(* IEC 61131-3 sources: A_BST22/ (part 2) *)

(* ---- simon_says_ladder_logic.st ---- *)
(*
Simon Says Game - Ladder Logic Implementation
Phase 1: 3 Buttons (Red, Blue, Yellow)
For Omron NX102-1100 PLC with Sysmac Studio

Author: Assistant
Date: 2025-10-01
Version: 1.0
*)

PROGRAM SimonSaysGame
VAR
    // Local working variables
    i : INT;
    ButtonPressed : INT;
    SequenceMatch : BOOL;
END_VAR

(* ========================================
   RUNG 1: INPUT MAPPING AND EDGE DETECTION
   ======================================== *)

// Map physical inputs to variables
RedButton_Input := %IX0.5;      // DI5
BlueButton_Input := %IX0.3;     // DI3
YellowButton_Input := %IX0.1;   // DI1

// Edge detection for button presses
RedButton_Rising := RedButton_Input AND NOT RedButton_Prev;
BlueButton_Rising := BlueButton_Input AND NOT BlueButton_Prev;
YellowButton_Rising := YellowButton_Input AND NOT YellowButton_Prev;

// Store previous states
RedButton_Prev := RedButton_Input;
BlueButton_Prev := BlueButton_Input;
YellowButton_Prev := YellowButton_Input;

(* ========================================
   RUNG 2: GAME INITIALIZATION
   ======================================== *)

// Initialize game on first scan or reset
IF FIRST_SCAN OR GameReset THEN
    GameState := 0;             // Idle state
    GameActive := FALSE;
    CurrentLevel := 1;
    SequenceLength := 1;
    PlaybackIndex := 0;
    InputIndex := 1;
    GameReset := FALSE;

    // Clear sequence array
    FOR i := 1 TO MaxLevel DO
        GameSequence[i] := 0;
    END_FOR;

    // Initialize random seed with system time
    RandomSeed := DWORD_TO_TIME(TIME());
END_IF;

(* ========================================
   RUNG 3: GAME START TRIGGER
   ======================================== *)

// Start game when any button is pressed in idle state
IF GameState = 0 AND (RedButton_Rising OR BlueButton_Rising OR YellowButton_Rising) THEN
    GameState := 1;             // Generate new sequence
    GameActive := TRUE;
    CurrentLevel := 1;
    SequenceLength := 1;
    GameWon := FALSE;
    GameLost := FALSE;
END_IF;

(* ========================================
   RUNG 4: RANDOM SEQUENCE GENERATION
   ======================================== *)

// Generate new sequence element
IF GameState = 1 THEN
    // Simple linear congruential generator for random numbers
    RandomValue := (RandomSeed * 1103515245 + 12345) MOD 16#7FFFFFFF;
    RandomSeed := RandomValue;

    // Convert to button number (1=Red, 2=Blue, 3=Yellow)
    NextButton := (INT(RandomValue MOD 3)) + 1;

    // Add to sequence
    GameSequence[SequenceLength] := NextButton;

    // Move to playback state
    GameState := 2;
    PlaybackIndex := 1;
    PlaybackActive := TRUE;

    // Start first flash timer
    FlashTimer.IN := TRUE;
    FlashTimer.PT := FLASH_TIME;
END_IF;

(* ========================================
   RUNG 5: SEQUENCE PLAYBACK LOGIC
   ======================================== *)

// Handle LED flashing during playback
IF GameState = 2 AND PlaybackActive THEN

    // Flash current button in sequence
    CASE GameSequence[PlaybackIndex] OF
        1: RedLED_Output := FlashTimer.IN AND NOT FlashTimer.Q;      // Red
        2: BlueLED_Output := FlashTimer.IN AND NOT FlashTimer.Q;     // Blue
        3: YellowLED_Output := FlashTimer.IN AND NOT FlashTimer.Q;   // Yellow
    END_CASE;

    // When flash timer expires, start gap timer
    IF FlashTimer.Q THEN
        FlashTimer.IN := FALSE;
        GapTimer.IN := TRUE;
        GapTimer.PT := GAP_TIME;

        // Turn off all LEDs during gap
        RedLED_Output := FALSE;
        BlueLED_Output := FALSE;
        YellowLED_Output := FALSE;
    END_IF;

    // When gap timer expires, move to next button or finish playback
    IF GapTimer.Q THEN
        GapTimer.IN := FALSE;
        PlaybackIndex := PlaybackIndex + 1;

        IF PlaybackIndex > SequenceLength THEN
            // Playback complete, start input phase
            PlaybackActive := FALSE;
            GameState := 3;
            InputIndex := 1;
            InputTimer.IN := TRUE;
            InputTimer.PT := INPUT_TIMEOUT;
        ELSE
            // Start next flash
            FlashTimer.IN := TRUE;
            FlashTimer.PT := FLASH_TIME;
        END_IF;
    END_IF;
END_IF;

// Call timer function blocks
FlashTimer();
GapTimer();

(* ========================================
   RUNG 6: PLAYER INPUT HANDLING
   ======================================== *)

// Handle player input during input phase
IF GameState = 3 THEN

    // Determine which button was pressed
    ButtonPressed := 0;
    IF RedButton_Rising THEN
        ButtonPressed := 1;
        LastButtonPressed := 1;
    ELSIF BlueButton_Rising THEN
        ButtonPressed := 2;
        LastButtonPressed := 2;
    ELSIF YellowButton_Rising THEN
        ButtonPressed := 3;
        LastButtonPressed := 3;
    END_IF;

    // Process button press
    IF ButtonPressed > 0 THEN
        // Check if correct button
        IF ButtonPressed = GameSequence[InputIndex] THEN
            CorrectSequence := TRUE;
            InputIndex := InputIndex + 1;

            // Reset input timer for next button
            InputTimer.IN := FALSE;
            InputTimer.IN := TRUE;
            InputTimer.PT := INPUT_TIMEOUT;

            // Check if sequence complete
            IF InputIndex > SequenceLength THEN
                // Level complete!
                GameState := 4;  // Success state
                SuccessTimer.IN := TRUE;
                SuccessTimer.PT := SUCCESS_DELAY;
            END_IF;
        ELSE
            // Wrong button - game over
            CorrectSequence := FALSE;
            GameState := 5;  // Fail state
            GameLost := TRUE;
        END_IF;
    END_IF;

    // Check for input timeout
    IF InputTimer.Q THEN
        GameState := 5;  // Fail state
        GameLost := TRUE;
        InputTimeout := TRUE;
    END_IF;

    InputTimer();
END_IF;

(* ========================================
   RUNG 7: SUCCESS HANDLING
   ======================================== *)

// Handle successful level completion
IF GameState = 4 THEN

    // Flash all LEDs to indicate success
    RedLED_Output := TRUE;
    BlueLED_Output := TRUE;
    YellowLED_Output := TRUE;

    // When success timer expires, advance to next level
    IF SuccessTimer.Q THEN
        SuccessTimer.IN := FALSE;
        CurrentLevel := CurrentLevel + 1;
        SequenceLength := SequenceLength + 1;

        // Check if game won (max level reached)
        IF CurrentLevel > MaxLevel THEN
            GameWon := TRUE;
            GameState := 0;  // Return to idle
            GameActive := FALSE;
        ELSE
            // Generate next level
            GameState := 1;
        END_IF;

        // Turn off success LEDs
        RedLED_Output := FALSE;
        BlueLED_Output := FALSE;
        YellowLED_Output := FALSE;
    END_IF;

    SuccessTimer();
END_IF;

(* ========================================
   RUNG 8: FAILURE HANDLING
   ======================================== *)

// Handle game failure
IF GameState = 5 THEN

    // Flash all LEDs rapidly to indicate failure
    IF (TIME() MOD T#200ms) < T#100ms THEN
        RedLED_Output := TRUE;
        BlueLED_Output := TRUE;
        YellowLED_Output := TRUE;
    ELSE
        RedLED_Output := FALSE;
        BlueLED_Output := FALSE;
        YellowLED_Output := FALSE;
    END_IF;

    // Auto-reset after 3 seconds
    IF NOT SuccessTimer.IN THEN
        SuccessTimer.IN := TRUE;
        SuccessTimer.PT := T#3000ms;
    END_IF;

    IF SuccessTimer.Q THEN
        GameReset := TRUE;
        SuccessTimer.IN := FALSE;
    END_IF;

    SuccessTimer();
END_IF;

(* ========================================
   RUNG 9: OUTPUT MAPPING
   ======================================== *)

// Map LED outputs to physical outputs
%QX0.0 := RedLED_Output;        // DO0
%QX0.1 := BlueLED_Output;       // DO1
%QX0.2 := YellowLED_Output;     // DO2

(* ========================================
   RUNG 10: STATUS AND DEBUG
   ======================================== *)

// Update debug status string
CASE GameState OF
    0: DebugState := 'IDLE - Press any button to start';
    1: DebugState := 'GENERATING sequence';
    2: DebugState := 'PLAYBACK - Watch the sequence';
    3: DebugState := 'INPUT - Repeat the sequence';
    4: DebugState := 'SUCCESS - Level complete!';
    5: DebugState := 'FAILED - Game over';
END_CASE;

// Test mode - all LEDs on (for testing)
IF AllLEDs_Test THEN
    %QX0.0 := TRUE;  // Red LED
    %QX0.1 := TRUE;  // Blue LED
    %QX0.2 := TRUE;  // Yellow LED
END_IF;

END_PROGRAM

(* ---- SimonSays.st ---- *)
// MAIN is N.C. → LED on when pressed
OLED_MAIN := NOT IBTN_MAIN;

// Color buttons → LED (when not in sequence display mode)
IF NOT SeqDisplay_Active THEN
    OLED_B := IBTN_B;
    OLED_R := IBTN_R;
    OLED_Y := IBTN_Y;
END_IF;

//  main game logic
Trig_Start(Clk := IBTN_B, Q => B);

IF B THEN
    Rand_Gen(Execute := TRUE, Seed := 0, Rnd => RandN);

    IF RandN < 0.333 THEN
        L_N := 1;  // Yellow
    ELSIF RandN < 0.666 THEN
        L_N := 2;  // Blue
    ELSE
        L_N := 3;  // Red
    END_IF;

    IF WriteIndex >= 50 THEN
        WriteIndex := 0;
        ArrayFull := TRUE;
    ELSIF WriteIndex < 0 THEN
        WriteIndex := 0;
    END_IF;

    Idx := TO_INT(WriteIndex);
    GameFlow_SN[Idx] := L_N;
    WriteIndex := WriteIndex + 1;

    // Trigger sequence display after adding new number
    SeqDisplay_Active := TRUE;
    SeqDisplay_Index := 0;
    SeqDisplay_Step := 0;  // 0 = LED ON, 1 = LED OFF
    T_SeqDisplay(IN := FALSE, PT := T#300ms);
END_IF;

// --- Sequence Display Logic ---
IF SeqDisplay_Active THEN
    IF NOT T_SeqDisplay.Q THEN
        T_SeqDisplay(IN := TRUE, PT := T#300ms);
    ELSE
        T_SeqDisplay(IN := FALSE, PT := T#300ms);
    END_IF;

    Trig_SeqTick(CLK := T_SeqDisplay.Q);
    SeqDisplay_Tick := Trig_SeqTick.Q;

    IF SeqDisplay_Tick THEN
        IF SeqDisplay_Step = 0 THEN
            // LED ON - display current sequence element
            CASE GameFlow_SN[SeqDisplay_Index] OF
                1:  OLED_Y := TRUE;  OLED_B := FALSE; OLED_R := FALSE;  // Yellow
                2:  OLED_Y := FALSE; OLED_B := TRUE;  OLED_R := FALSE;  // Blue
                3:  OLED_Y := FALSE; OLED_B := FALSE; OLED_R := TRUE;   // Red
                ELSE
                    OLED_Y := FALSE; OLED_B := FALSE; OLED_R := FALSE;
            END_CASE;
            SeqDisplay_Step := 1;
        ELSE
            // LED OFF - pause between elements
            OLED_Y := FALSE; OLED_B := FALSE; OLED_R := FALSE;
            SeqDisplay_Step := 0;
            SeqDisplay_Index := SeqDisplay_Index + 1;

            // Check if we've displayed the entire sequence
            IF SeqDisplay_Index >= WriteIndex THEN
                SeqDisplay_Active := FALSE;
                OLED_Y := FALSE; OLED_B := FALSE; OLED_R := FALSE;
            END_IF;
        END_IF;
    END_IF;
END_IF;

// -auto-reset edge when WriteIndex hits 50
Trig_Wrap(CLK := (WriteIndex = 50));
ResetReq := RI OR Trig_Wrap.Q;      // manual RI or auto edge at 50
Trig_Reset(CLK := ResetReq);

IF Trig_Reset.Q THEN
    AryAddV(In1 := GameFlow_S[0], In2 := L_N, Size := 50, AryOut := GameFlow_SN[0]);

    GameOver_Active := TRUE;
    GameOver_Step := -1;
    T_Seq(IN := FALSE, PT := T#300ms);

    WriteIndex := 0;
    ArrayFull := TRUE;
END_IF;

// --- game over LED sequence (R -> B -> Y, once) ---
IF GameOver_Active THEN
    IF NOT T_Seq.Q THEN
        T_Seq(IN := TRUE, PT := T#300ms);
    ELSE
        T_Seq(IN := FALSE, PT := T#300ms);
    END_IF;

    Trig_Tick(CLK := T_Seq.Q);
    GameOver_Tick := Trig_Tick.Q;

    IF GameOver_Tick THEN
        GameOver_Step := GameOver_Step + 1;
    END_IF;

    CASE GameOver_Step OF
        0:  OLED_R := TRUE;  OLED_B := FALSE; OLED_Y := FALSE;
        1:  OLED_R := FALSE; OLED_B := TRUE;  OLED_Y := FALSE;
        2:  OLED_R := FALSE; OLED_B := FALSE; OLED_Y := TRUE;
        4:  OLED_R := FALSE; OLED_B := FALSE; OLED_Y := FALSE;
        5:  OLED_R := TRUE;  OLED_B := TRUE;  OLED_Y := TRUE;
        6:  OLED_R := FALSE; OLED_B := FALSE; OLED_Y := FALSE;
        7:  OLED_R := TRUE;  OLED_B := TRUE;  OLED_Y := TRUE;
        ELSE
            OLED_R := FALSE; OLED_B := FALSE; OLED_Y := FALSE;
    END_CASE;

    IF GameOver_Step > 7 THEN
        GameOver_Active := FALSE;
        OLED_R := FALSE; OLED_B := FALSE; OLED_Y := FALSE;
    END_IF;
END_IF;

(* ---- SimonSays_Phase1.st ---- *)
(* ====================================================================
   SIMON SAYS GAME - PHASE 1 (3 BUTTONS)
   For Omron NX102-1100 PLC

   Hardware Configuration:
   - Yellow Button: DI1 (input), DO2 (LED)
   - Blue Button:   DI3 (input), DO1 (LED)
   - Red Button:    DI5 (input), DO0 (LED)

   Author: PLC Programming Assistant
   Date: October 2025
   Version: 1.0
   ==================================================================== *)

PROGRAM SimonSays_Phase1
VAR
    (* ==================== INPUT MAPPING ==================== *)
    Yellow_Button_Input AT %IX0.1 : BOOL;  (* DI1 - Yellow button press *)
    Blue_Button_Input   AT %IX0.3 : BOOL;  (* DI3 - Blue button press *)
    Red_Button_Input    AT %IX0.5 : BOOL;  (* DI5 - Red button press *)

    (* ==================== OUTPUT MAPPING ==================== *)
    Red_LED_Output      AT %QX0.0 : BOOL;  (* DO0 - Red LED *)
    Blue_LED_Output     AT %QX0.1 : BOOL;  (* DO1 - Blue LED *)
    Yellow_LED_Output   AT %QX0.2 : BOOL;  (* DO2 - Yellow LED *)

    (* ==================== GAME STATE MACHINE ==================== *)
    GameState           : INT := 0;        (* 0=Idle, 1=StartNewGame, 2=ShowSequence, 3=WaitForPlayer, 4=CheckInput, 5=GameOver, 6=Victory *)

    (* ==================== SEQUENCE MANAGEMENT ==================== *)
    GameSequence        : ARRAY[0..49] OF INT := [50(0)];  (* Stores the sequence (1=Yellow, 2=Blue, 3=Red) *)
    CurrentLevel        : INT := 0;        (* Current level/length of sequence *)
    SequenceIndex       : INT := 0;        (* Index for displaying/checking sequence *)
    PlayerInputIndex    : INT := 0;        (* Current position in player input *)
    MaxLevel            : INT := 10;       (* Maximum sequence length *)

    (* ==================== TIMING CONTROLS ==================== *)
    FlashTimer          : TON;              (* Timer for LED flash duration *)
    GapTimer            : TON;              (* Timer for gap between flashes *)
    InputTimeoutTimer   : TON;              (* Timer for player input timeout *)
    StartDelayTimer     : TON;              (* Timer for game start delay *)

    FlashTime           : TIME := T#500MS;  (* LED on duration *)
    GapTime             : TIME := T#300MS;  (* Gap between LED flashes *)
    InputTimeout        : TIME := T#5S;     (* Player input timeout *)
    StartDelay          : TIME := T#2S;     (* Delay before starting game *)

    (* ==================== PLAYER INPUT HANDLING ==================== *)
    LastButtonPressed   : INT := 0;        (* Last button pressed by player *)
    ButtonPressDetected : BOOL := FALSE;   (* Flag for button press detection *)
    InputCorrect        : BOOL := TRUE;    (* Flag for correct input *)

    (* ==================== EDGE DETECTION ==================== *)
    Yellow_Button_Edge  : R_TRIG;          (* Rising edge detection for Yellow *)
    Blue_Button_Edge    : R_TRIG;          (* Rising edge detection for Blue *)
    Red_Button_Edge     : R_TRIG;          (* Rising edge detection for Red *)

    (* ==================== RANDOM NUMBER GENERATION ==================== *)
    RandomSeed          : DINT := 12345;   (* Seed for random number *)
    RandomValue         : INT;             (* Generated random value *)

    (* ==================== CONTROL FLAGS ==================== *)
    StartGame           : BOOL := FALSE;   (* Start game trigger *)
    ResetGame           : BOOL := FALSE;   (* Reset game trigger *)
    ShowingSequence     : BOOL := FALSE;   (* Flag indicating sequence display *)
    WaitingForInput     : BOOL := FALSE;   (* Flag indicating waiting for player *)

END_VAR

(* ==================== MAIN PROGRAM LOGIC ==================== *)

(* Edge detection for button inputs *)
Yellow_Button_Edge(CLK := Yellow_Button_Input);
Blue_Button_Edge(CLK := Blue_Button_Input);
Red_Button_Edge(CLK := Red_Button_Input);

(* ==================== GAME STATE MACHINE ==================== *)
CASE GameState OF

    0: (* IDLE STATE - Waiting to start *)
        (* Reset all LEDs *)
        Yellow_LED_Output := FALSE;
        Blue_LED_Output := FALSE;
        Red_LED_Output := FALSE;

        (* Reset game variables *)
        CurrentLevel := 0;
        SequenceIndex := 0;
        PlayerInputIndex := 0;
        ShowingSequence := FALSE;
        WaitingForInput := FALSE;

        (* Check for start trigger - any button press starts the game *)
        IF Yellow_Button_Edge.Q OR Blue_Button_Edge.Q OR Red_Button_Edge.Q THEN
            StartGame := TRUE;
        END_IF;

        IF StartGame THEN
            GameState := 1;  (* Move to StartNewGame *)
            StartGame := FALSE;
        END_IF;

    1: (* START NEW GAME / ADD TO SEQUENCE *)
        (* Flash all LEDs to indicate new round *)
        StartDelayTimer(IN := TRUE, PT := StartDelay);

        Yellow_LED_Output := TRUE;
        Blue_LED_Output := TRUE;
        Red_LED_Output := TRUE;

        IF StartDelayTimer.Q THEN
            StartDelayTimer(IN := FALSE);

            (* Turn off all LEDs *)
            Yellow_LED_Output := FALSE;
            Blue_LED_Output := FALSE;
            Red_LED_Output := FALSE;

            (* Add new random element to sequence *)
            CurrentLevel := CurrentLevel + 1;

            (* Generate random number 1-3 *)
            RandomSeed := (RandomSeed * 1103515245 + 12345) MOD 2147483648;
            RandomValue := (ABS(RandomSeed) MOD 3) + 1;
            GameSequence[CurrentLevel - 1] := RandomValue;

            (* Reset indices *)
            SequenceIndex := 0;
            PlayerInputIndex := 0;

            (* Move to show sequence *)
            GameState := 2;
        END_IF;

    2: (* SHOW SEQUENCE - Display pattern to player *)
        ShowingSequence := TRUE;
        WaitingForInput := FALSE;

        (* Display current element in sequence *)
        IF SequenceIndex < CurrentLevel THEN

            (* Flash the appropriate LED *)
            IF NOT FlashTimer.IN AND NOT GapTimer.IN THEN
                (* Start flash *)
                FlashTimer(IN := TRUE, PT := FlashTime);

                (* Turn on appropriate LED *)
                CASE GameSequence[SequenceIndex] OF
                    1: Yellow_LED_Output := TRUE;
                    2: Blue_LED_Output := TRUE;
                    3: Red_LED_Output := TRUE;
                END_CASE;
            END_IF;

            (* Handle flash timing *)
            FlashTimer(IN := FlashTimer.IN, PT := FlashTime);
            IF FlashTimer.Q THEN
                (* Turn off all LEDs *)
                Yellow_LED_Output := FALSE;
                Blue_LED_Output := FALSE;
                Red_LED_Output := FALSE;

                FlashTimer(IN := FALSE);

                (* Start gap timer *)
                GapTimer(IN := TRUE, PT := GapTime);
            END_IF;

            (* Handle gap timing *)
            GapTimer(IN := GapTimer.IN, PT := GapTime);
            IF GapTimer.Q THEN
                GapTimer(IN := FALSE);

                (* Move to next element *)
                SequenceIndex := SequenceIndex + 1;
            END_IF;

        ELSE
            (* Sequence display complete *)
            ShowingSequence := FALSE;
            PlayerInputIndex := 0;
            GameState := 3;  (* Move to wait for player *)
        END_IF;

    3: (* WAIT FOR PLAYER INPUT *)
        WaitingForInput := TRUE;
        ShowingSequence := FALSE;

        (* Start input timeout timer *)
        InputTimeoutTimer(IN := TRUE, PT := InputTimeout);

        (* Check for button presses *)
        ButtonPressDetected := FALSE;
        LastButtonPressed := 0;

        IF Yellow_Button_Edge.Q THEN
            ButtonPressDetected := TRUE;
            LastButtonPressed := 1;
            Yellow_LED_Output := TRUE;  (* Light up while pressed *)
        ELSIF Blue_Button_Edge.Q THEN
            ButtonPressDetected := TRUE;
            LastButtonPressed := 2;
            Blue_LED_Output := TRUE;    (* Light up while pressed *)
        ELSIF Red_Button_Edge.Q THEN
            ButtonPressDetected := TRUE;
            LastButtonPressed := 3;
            Red_LED_Output := TRUE;     (* Light up while pressed *)
        END_IF;

        (* Turn off LEDs when buttons are released *)
        IF NOT Yellow_Button_Input THEN
            Yellow_LED_Output := FALSE;
        END_IF;
        IF NOT Blue_Button_Input THEN
            Blue_LED_Output := FALSE;
        END_IF;
        IF NOT Red_Button_Input THEN
            Red_LED_Output := FALSE;
        END_IF;

        (* Process button press *)
        IF ButtonPressDetected THEN
            InputTimeoutTimer(IN := FALSE);  (* Reset timeout *)
            GameState := 4;  (* Move to check input *)
        END_IF;

        (* Check for timeout *)
        IF InputTimeoutTimer.Q THEN
            InputTimeoutTimer(IN := FALSE);
            GameState := 5;  (* Game over - timeout *)
        END_IF;

    4: (* CHECK PLAYER INPUT *)
        (* Verify if the input matches the sequence *)
        IF LastButtonPressed = GameSequence[PlayerInputIndex] THEN
            (* Correct input *)
            PlayerInputIndex := PlayerInputIndex + 1;

            IF PlayerInputIndex >= CurrentLevel THEN
                (* Player completed the sequence *)
                IF CurrentLevel >= MaxLevel THEN
                    GameState := 6;  (* Victory! *)
                ELSE
                    (* Add delay before next round *)
                    StartDelayTimer(IN := TRUE, PT := T#1S);
                    IF StartDelayTimer.Q THEN
                        StartDelayTimer(IN := FALSE);
                        GameState := 1;  (* Next level *)
                    END_IF;
                END_IF;
            ELSE
                (* Wait for next input *)
                GameState := 3;
            END_IF;
        ELSE
            (* Wrong input *)
            GameState := 5;  (* Game over *)
        END_IF;

    5: (* GAME OVER *)
        (* Flash red LED to indicate failure *)
        FlashTimer(IN := TRUE, PT := T#200MS);

        IF FlashTimer.Q THEN
            Red_LED_Output := NOT Red_LED_Output;
            FlashTimer(IN := FALSE);
        END_IF;

        (* Wait for button press to restart *)
        IF Yellow_Button_Edge.Q OR Blue_Button_Edge.Q OR Red_Button_Edge.Q THEN
            FlashTimer(IN := FALSE);
            GameState := 0;  (* Return to idle *)
        END_IF;

    6: (* VICTORY *)
        (* Celebration pattern - cycle through all LEDs *)
        FlashTimer(IN := TRUE, PT := T#100MS);

        IF FlashTimer.Q THEN
            FlashTimer(IN := FALSE);

            (* Rotate LEDs *)
            IF Yellow_LED_Output AND NOT Blue_LED_Output AND NOT Red_LED_Output THEN
                Yellow_LED_Output := FALSE;
                Blue_LED_Output := TRUE;
            ELSIF Blue_LED_Output AND NOT Red_LED_Output THEN
                Blue_LED_Output := FALSE;
                Red_LED_Output := TRUE;
            ELSIF Red_LED_Output THEN
                Red_LED_Output := FALSE;
                Yellow_LED_Output := TRUE;
            ELSE
                Yellow_LED_Output := TRUE;
            END_IF;
        END_IF;

        (* Wait for button press to restart *)
        IF Yellow_Button_Edge.Q OR Blue_Button_Edge.Q OR Red_Button_Edge.Q THEN
            FlashTimer(IN := FALSE);
            GameState := 0;  (* Return to idle *)
        END_IF;

END_CASE;

END_PROGRAM

(* ---- SimonSays_Phase1_Main.st ---- *)
(* ====================================================================== *)
(* Simon Says Game - Phase 1 (3 Buttons)                                 *)
(* For Omron NX102-1100 PLC                                             *)
(* Version: 1.0                                                          *)
(* Date: October 2025                                                    *)
(* ====================================================================== *)

(* ====================================================================== *)
(* I/O MAPPING                                                           *)
(* ====================================================================== *)
(* INPUTS (NX-ID4442):
   DI1 - Yellow Button Contact (Pin 4, Black wire)
   DI3 - Blue Button Contact (Pin 4, Black wire)
   DI5 - Red Button Contact (Pin 4, Black wire)

   OUTPUTS (NX-OD4256):
   DO0 - Red Button LED (Pin 2, White wire)
   DO1 - Blue Button LED (Pin 2, White wire)
   DO2 - Yellow Button LED (Pin 2, White wire)
*)

(* ====================================================================== *)
(* VARIABLE DECLARATIONS                                                 *)
(* ====================================================================== *)

VAR_GLOBAL
    (* Physical I/O *)
    YellowButton_Input AT %IX0.1 : BOOL;    (* DI1 *)
    BlueButton_Input AT %IX0.3 : BOOL;      (* DI3 *)
    RedButton_Input AT %IX0.5 : BOOL;       (* DI5 *)

    RedButton_LED AT %QX0.0 : BOOL;         (* DO0 *)
    BlueButton_LED AT %QX0.1 : BOOL;        (* DO1 *)
    YellowButton_LED AT %QX0.2 : BOOL;      (* DO2 *)

    (* Game State Machine *)
    GameState : INT := 0;
    (* 0 = IDLE/WAITING
       1 = SHOW_SEQUENCE
       2 = WAIT_FOR_INPUT
       3 = GAME_OVER_WIN
       4 = GAME_OVER_LOSE *)

    (* Game Control *)
    GameStart : BOOL := FALSE;
    GameReset : BOOL := FALSE;
    StartButton : BOOL := FALSE;  (* Will be mapped to selector switch later *)

    (* Sequence Storage *)
    GameSequence : ARRAY[0..49] OF INT;     (* Store up to 50 moves *)
    CurrentLevel : INT := 0;                (* Current game level/length *)
    SequenceIndex : INT := 0;                (* Current position in sequence *)
    PlayerInputIndex : INT := 0;             (* Player's current input position *)
    MaxLevel : INT := 10;                    (* Maximum sequence length *)

    (* Player Input *)
    PlayerInput : INT := 0;                  (* Current button pressed by player *)
    LastPlayerInput : INT := 0;              (* Previous input for edge detection *)
    InputCorrect : BOOL := TRUE;             (* Track if player input is correct *)

    (* Timing *)
    ShowTimer : TON;                         (* Timer for showing each LED *)
    GapTimer : TON;                          (* Timer for gap between LEDs *)
    InputTimer : TON;                        (* Timer for player input timeout *)
    GameOverTimer : TON;                     (* Timer for game over display *)

    ShowTime : TIME := T#500MS;             (* Time to show each LED *)
    GapTime : TIME := T#200MS;              (* Gap between LEDs *)
    InputTimeout : TIME := T#3S;            (* Player input timeout *)
    GameOverTime : TIME := T#2S;            (* Game over display time *)

    (* Random Number Generation *)
    RandomSeed : DINT := 0;
    RandomValue : INT := 0;

    (* Edge Detection *)
    YellowButton_Rising : R_TRIG;
    BlueButton_Rising : R_TRIG;
    RedButton_Rising : R_TRIG;
    StartButton_Rising : R_TRIG;

    (* Flags *)
    ShowingLED : BOOL := FALSE;
    WaitingGap : BOOL := FALSE;
    SequenceComplete : BOOL := FALSE;
    InputReceived : BOOL := FALSE;

END_VAR

(* ====================================================================== *)
(* MAIN PROGRAM                                                          *)
(* ====================================================================== *)

PROGRAM SimonSaysMain

    (* Edge Detection for Buttons *)
    YellowButton_Rising(CLK := YellowButton_Input);
    BlueButton_Rising(CLK := BlueButton_Input);
    RedButton_Rising(CLK := RedButton_Input);
    StartButton_Rising(CLK := StartButton);

    (* Random Seed Update - Use system time or counter *)
    RandomSeed := RandomSeed + 1;
    IF RandomSeed > 1000000 THEN
        RandomSeed := 0;
    END_IF;

    (* ====================================================================== *)
    (* GAME STATE MACHINE                                                    *)
    (* ====================================================================== *)

    CASE GameState OF

        (* ------------------------------------------------------------ *)
        0: (* IDLE/WAITING STATE *)
        (* ------------------------------------------------------------ *)
            (* Reset all LEDs *)
            RedButton_LED := FALSE;
            BlueButton_LED := FALSE;
            YellowButton_LED := FALSE;

            (* Reset game variables *)
            CurrentLevel := 0;
            SequenceIndex := 0;
            PlayerInputIndex := 0;
            InputCorrect := TRUE;
            ShowingLED := FALSE;
            WaitingGap := FALSE;

            (* Wait for start signal *)
            IF StartButton_Rising.Q OR GameStart THEN
                GameStart := FALSE;
                (* Initialize first sequence *)
                CurrentLevel := 1;
                (* Generate first random button (1=Yellow, 2=Blue, 3=Red) *)
                RandomValue := INT(RandomSeed MOD 3) + 1;
                GameSequence[0] := RandomValue;
                (* Move to show sequence state *)
                GameState := 1;
                SequenceIndex := 0;
            END_IF;

        (* ------------------------------------------------------------ *)
        1: (* SHOW_SEQUENCE STATE *)
        (* ------------------------------------------------------------ *)
            (* Display the current sequence to the player *)

            IF NOT ShowingLED AND NOT WaitingGap THEN
                (* Start showing next LED in sequence *)
                IF SequenceIndex < CurrentLevel THEN
                    ShowingLED := TRUE;
                    ShowTimer(IN := FALSE);
                    ShowTimer(IN := TRUE, PT := ShowTime);
                ELSE
                    (* Sequence complete, move to input state *)
                    SequenceComplete := TRUE;
                    GameState := 2;
                    PlayerInputIndex := 0;
                    InputTimer(IN := FALSE);
                    InputTimer(IN := TRUE, PT := InputTimeout);
                END_IF;
            END_IF;

            (* Show LED based on sequence *)
            IF ShowingLED THEN
                ShowTimer(IN := TRUE, PT := ShowTime);

                (* Turn on appropriate LED *)
                CASE GameSequence[SequenceIndex] OF
                    1: YellowButton_LED := TRUE;
                    2: BlueButton_LED := TRUE;
                    3: RedButton_LED := TRUE;
                END_CASE;

                (* Check if show time expired *)
                IF ShowTimer.Q THEN
                    (* Turn off all LEDs *)
                    RedButton_LED := FALSE;
                    BlueButton_LED := FALSE;
                    YellowButton_LED := FALSE;

                    ShowingLED := FALSE;
                    WaitingGap := TRUE;
                    GapTimer(IN := FALSE);
                    GapTimer(IN := TRUE, PT := GapTime);
                END_IF;
            END_IF;

            (* Gap between LEDs *)
            IF WaitingGap THEN
                GapTimer(IN := TRUE, PT := GapTime);

                IF GapTimer.Q THEN
                    WaitingGap := FALSE;
                    SequenceIndex := SequenceIndex + 1;
                END_IF;
            END_IF;

        (* ------------------------------------------------------------ *)
        2: (* WAIT_FOR_INPUT STATE *)
        (* ------------------------------------------------------------ *)
            (* Wait for player to repeat the sequence *)

            (* Update input timeout timer *)
            InputTimer(IN := TRUE, PT := InputTimeout);

            (* Check for timeout *)
            IF InputTimer.Q THEN
                (* Player took too long - game over *)
                GameState := 4; (* GAME_OVER_LOSE *)
                GameOverTimer(IN := FALSE);
                GameOverTimer(IN := TRUE, PT := GameOverTime);
            END_IF;

            (* Check for button presses *)
            InputReceived := FALSE;
            PlayerInput := 0;

            IF YellowButton_Rising.Q THEN
                PlayerInput := 1;
                InputReceived := TRUE;
                YellowButton_LED := TRUE;
            ELSIF BlueButton_Rising.Q THEN
                PlayerInput := 2;
                InputReceived := TRUE;
                BlueButton_LED := TRUE;
            ELSIF RedButton_Rising.Q THEN
                PlayerInput := 3;
                InputReceived := TRUE;
                RedButton_LED := TRUE;
            END_IF;

            (* Turn off LED when button is released *)
            IF NOT YellowButton_Input THEN
                YellowButton_LED := FALSE;
            END_IF;
            IF NOT BlueButton_Input THEN
                BlueButton_LED := FALSE;
            END_IF;
            IF NOT RedButton_Input THEN
                RedButton_LED := FALSE;
            END_IF;

            (* Process input if received *)
            IF InputReceived THEN
                (* Reset timeout timer *)
                InputTimer(IN := FALSE);
                InputTimer(IN := TRUE, PT := InputTimeout);

                (* Check if input matches sequence *)
                IF PlayerInput = GameSequence[PlayerInputIndex] THEN
                    (* Correct input *)
                    PlayerInputIndex := PlayerInputIndex + 1;

                    (* Check if player completed current sequence *)
                    IF PlayerInputIndex >= CurrentLevel THEN
                        (* Sequence completed successfully *)
                        IF CurrentLevel >= MaxLevel THEN
                            (* Player wins! *)
                            GameState := 3; (* GAME_OVER_WIN *)
                        ELSE
                            (* Add next random button to sequence *)
                            CurrentLevel := CurrentLevel + 1;
                            RandomValue := INT((RandomSeed + CurrentLevel * 7) MOD 3) + 1;
                            GameSequence[CurrentLevel - 1] := RandomValue;

                            (* Wait a bit then show new sequence *)
                            GapTimer(IN := FALSE);
                            WaitingGap := TRUE;
                            GapTimer(IN := TRUE, PT := T#1S);

                            (* Return to show sequence state *)
                            GameState := 1;
                            SequenceIndex := 0;
                            ShowingLED := FALSE;
                        END_IF;
                    END_IF;
                ELSE
                    (* Wrong input - game over *)
                    GameState := 4; (* GAME_OVER_LOSE *)
                    GameOverTimer(IN := FALSE);
                    GameOverTimer(IN := TRUE, PT := GameOverTime);
                END_IF;
            END_IF;

        (* ------------------------------------------------------------ *)
        3: (* GAME_OVER_WIN STATE *)
        (* ------------------------------------------------------------ *)
            (* Flash all LEDs to indicate win *)
            GameOverTimer(IN := TRUE, PT := GameOverTime);

            (* Flash pattern for win *)
            IF (GameOverTimer.ET < T#200MS) OR
               ((GameOverTimer.ET >= T#400MS) AND (GameOverTimer.ET < T#600MS)) OR
               ((GameOverTimer.ET >= T#800MS) AND (GameOverTimer.ET < T#1S)) THEN
                RedButton_LED := TRUE;
                BlueButton_LED := TRUE;
                YellowButton_LED := TRUE;
            ELSE
                RedButton_LED := FALSE;
                BlueButton_LED := FALSE;
                YellowButton_LED := FALSE;
            END_IF;

            (* Return to idle after celebration *)
            IF GameOverTimer.Q THEN
                GameState := 0;
            END_IF;

        (* ------------------------------------------------------------ *)
        4: (* GAME_OVER_LOSE STATE *)
        (* ------------------------------------------------------------ *)
            (* Flash red LED to indicate loss *)
            GameOverTimer(IN := TRUE, PT := GameOverTime);

            (* Flash pattern for lose *)
            IF (GameOverTimer.ET < T#300MS) OR
               ((GameOverTimer.ET >= T#600MS) AND (GameOverTimer.ET < T#900MS)) OR
               ((GameOverTimer.ET >= T#1200MS) AND (GameOverTimer.ET < T#1500MS)) THEN
                RedButton_LED := TRUE;
            ELSE
                RedButton_LED := FALSE;
            END_IF;

            BlueButton_LED := FALSE;
            YellowButton_LED := FALSE;

            (* Return to idle after game over display *)
            IF GameOverTimer.Q THEN
                GameState := 0;
            END_IF;

    END_CASE;

    (* Manual Reset *)
    IF GameReset THEN
        GameState := 0;
        GameReset := FALSE;
    END_IF;

END_PROGRAM
